PROGRAM MAIN
VAR
	nContador AT %Q*: DINT;
END_VAR

nContador := nContador + 1;

END_PROGRAM

(* stored: Version 1.1.0.1, ProductVersion 3.1.4024.4
   POU MAIN: Id {bd2073ad-7f80-4a92-a7bb-c30c81baa107}, SpecialFunc None *)
